% RSLogix 500 project 9.3.RSS, saved by version 8.30.00.16 %
PROJECT "9.3"    % processor: Bul.1763 MicroLogix 1100 Series B %

PROGRAM FILES
  LAD 2   6 rungs

DATA FILES
  O0 OUTPUT  4 elements
  I1 INPUT  6 elements
  S2 STATUS  66 elements
  B3 BINARY  1 elements
  T4 TIMER  1 elements
  C5 COUNTER  3 elements
  R6 CONTROL  1 elements
  N7 INTEGER  2 elements
  F8 FLOAT  1 elements

LADDER 2
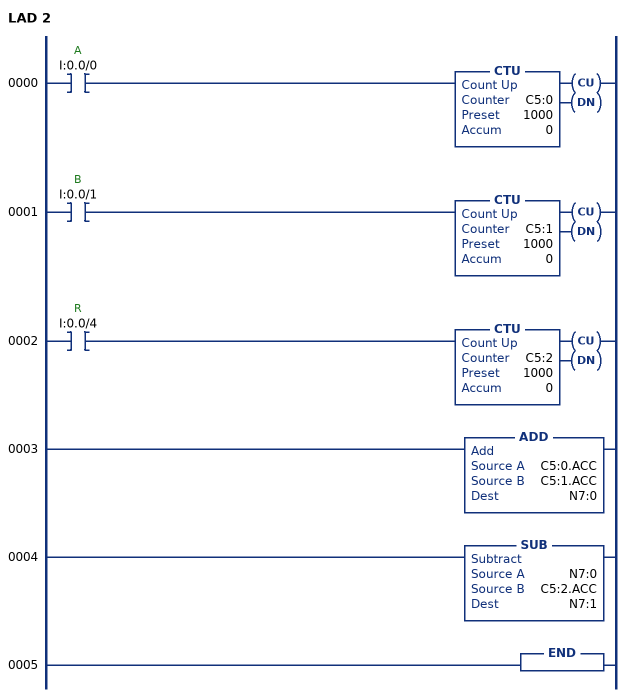
% Rung: 0 %
SOR XIC I:0.0/0 CTU C5:0 1000 0 EOR
%   I:0.0/0  "A" %
% Rung: 1 %
SOR XIC I:0.0/1 CTU C5:1 1000 0 EOR
%   I:0.0/1  "B" %
% Rung: 2 %
SOR XIC I:0.0/4 CTU C5:2 1000 0 EOR
%   I:0.0/4  "R" %
% Rung: 3 %
SOR ADD C5:0.ACC C5:1.ACC N7:0 EOR
% Rung: 4 %
SOR SUB N7:0 C5:2.ACC N7:1 EOR
% Rung: 5 %
SOR END EOR

OTHER DOCUMENTED ADDRESSES
  I:0.0/3  "C"

DATA TABLE (non-zero values as saved)
DATA C5
% .PRE .ACC %
% C5:0 % 1000 0
% C5:1 % 1000 0
% C5:2 % 1000 0
